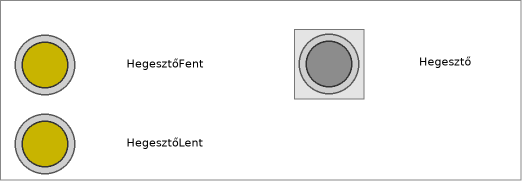
VISUALIZATION TempPistiHegesztes  // 522x181
    Lamp1 (10,30 70x70), variable: GVL.bHegeszto3Fent, style: Lamp-Lamp1-Yellow
    Label (90,49 150x30), "HegesztőFent"
    Lamp1 (10,109 70x70), variable: GVL.bHegeszto3Lent, style: Lamp-Lamp1-Yellow
    Label (90,128 150x30), "HegesztőLent"
    PushSwitch (294,29 70x70), variable: HEGESZTOK.bHegesztoFejekOutput[2], behaviour: TOGGLE, style: Switch-PushSwitch-Gray
    Label (370,47 150x30), "Hegesztő"
END_VISUALIZATION

(* stored: Version 1.1.0.1, ProductVersion 3.1.4024.11
   Visu TempPistiHegesztes: Id {a5eff718-b224-4ae9-a4f1-33a3ccae3e67} *)
